// TIA Portal project "Project44" (V11)

(* hardware
DEVICE "S7-400 station_1"  S7400.Device
   slot 0: "UR1_0"  UR1  6ES7 400-1TA01-0AA0
   slot 2: "PLC_1"  CPU 416F-3 PN/DP  6ES7 416-3FR05-0AB0  V5.3
      slot 5: "PROFINET interface_1"  PN-IO
         slot 1: "Port_1"  Port
         slot 2: "Port_2"  Port
*)

// ===== PLC "PLC_1"  CPU 416F-3 PN/DP =====

VAR_GLOBAL   // PLC tag table "Default tag table"
   "Tag_1" AT %I0.0 : Bool;
   "czerwone 5s" AT %M0.0 : Bool;
   "Tag_2" AT %M10.0 : Bool;
   "żółte i czerwone" AT %M0.1 : Bool;
   "Tag_3" AT %M10.1 : Bool;
   "zielone" AT %M0.2 : Bool;
   "Tag_4" AT %M10.2 : Bool;
   "żółte" AT %M0.3 : Bool;
   "Tag_5" AT %M10.3 : Bool;
   "czerwone" AT %M0.4 : Bool;
   "Tag_6" AT %M10.5 : Bool;
   "Tag_7" AT %M10.4 : Bool;
   "Tag_8" AT %M11.0 : Bool;
   "żółte i czerwone 2" AT %M0.5 : Bool;
   "Tag_9" AT %M11.1 : Bool;
   "zielone 2" AT %M0.6 : Bool;
   "Tag_10" AT %M9.0 : Bool;
   "Tag_11" AT %M11.2 : Bool;
   "żółte 2" AT %M0.7 : Bool;
   "Tag_12" AT %M11.3 : Bool;
   "czerwone 2" AT %M1.0 : Bool;
   "Tag_13" AT %M9.1 : Bool;
   "Tag_14" AT %M11.4 : Bool;
   "Tag_15" AT %M11.5 : Bool;
   "Tag_16" AT %M8.0 : Bool;
   "Tag_17" AT %M8.1 : Bool;
   "Tag_18" AT %M8.2 : Bool;
   "Tag_19" AT %M8.5 : Bool;
   "Tag_20" AT %M8.6 : Bool;
   "1 CZERWONE" AT %Q0.0 : Bool;
   "1 ŻÓŁTE" AT %Q0.1 : Bool;
   "1 ZIELONE" AT %Q0.2 : Bool;
   "2 CZERWONE" AT %Q0.3 : Bool;
   "2 ŻÓŁTE" AT %Q0.4 : Bool;
   "2 ZIELONE" AT %Q0.5 : Bool;
   "Tag_21" AT %M11.7 : Bool;
   "Tag_22" AT %M11.6 : Bool;
END_VAR

ORGANIZATION_BLOCK "Main"   // OB1, LAD
TITLE = "Main Program Sweep (Cycle)"
{ S7_Optimized_Access := 'FALSE' }
VERSION : 0.1
   VAR_TEMP
      OB1_EV_CLASS : Byte;   // Bits 0-3 = 1 (Coming event), Bits 4-7 = 1 (Event class 1)
      OB1_SCAN_1 : Byte;   // 1 (Cold restart scan 1 of OB 1), 3 (Scan 2-n of OB 1)
      OB1_PRIORITY : Byte;   // Priority of OB Execution
      OB1_OB_NUMBR : Byte;   // 1 (Organization block 1, OB1)
      OB1_RESERVED_1 : Byte;   // Reserved for system
      OB1_RESERVED_2 : Byte;   // Reserved for system
      OB1_PREV_CYCLE : Int;   // Cycle time of previous OB1 scan (milliseconds)
      OB1_MIN_CYCLE : Int;   // Minimum cycle time of OB1 (milliseconds)
      OB1_MAX_CYCLE : Int;   // Maximum cycle time of OB1 (milliseconds)
      OB1_DATE_TIME : Date_And_Time;   // Date and time OB1 started
   END_VAR
BEGIN
END_ORGANIZATION_BLOCK